FUNCTION_BLOCK Matrix_Inverse (* Template for a simple Basic Function Block Type *)
  (* Standard: 61499-2; Description: Calculates an Inverse of a matrix useing Gauss Jordan Elimination Method. *)
  (* Version 1.0, 2020-08-06, Hafiezd *)
  (* Version 1.1, 2020-08-12, Candra Wardaya *)
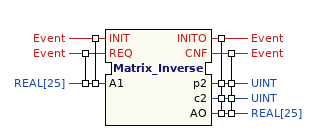
  EVENT_INPUT
    INIT WITH A1; (* Initialization Request *)
    REQ WITH A1; (* Normal Execution Request *)
  END_EVENT
  EVENT_OUTPUT
    INITO WITH AO, p2, c2; (* Initialization Confirm *)
    CNF WITH AO, p2, c2; (* Execution Confirmation *)
  END_EVENT
  VAR_INPUT
    A1 : ARRAY [0..24] OF REAL; (* Matrix Array Input *)
  END_VAR
  VAR_OUTPUT
    p2 : UINT; (* Output Row Size *)
    c2 : UINT; (* Output Column Size *)
    AO : ARRAY [0..24] OF REAL; (* Matrix Inverse Output Array *)
  END_VAR
  VAR
    i : UINT; (* Row Index *)
    j : UINT; (* Column Index *)
    c1 : UINT; (* Augmented Column Size *)
    B : ARRAY [0..99] OF REAL; (* Augmented Matrix of p * c_aug size *)
    ratio : REAL; (* zero-ing factor *)
    k : UINT; (* Augmented Column Index *)
    divisor : REAL; (* Identity factor *)
    p : UINT := 5; (* Internal Variable *)
    c : UINT := 5; (* Internal Variable *)
  END_VAR
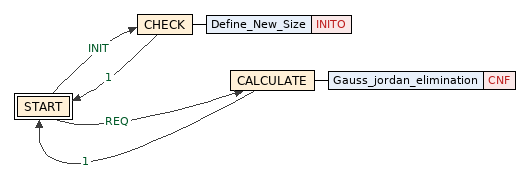
  EC_STATES
    START; (* Initial State *)
    CHECK : Define_New_Size -> INITO;
    CALCULATE : Gauss_jordan_elimination -> CNF;
  END_STATES
  EC_TRANSITIONS
    START TO CHECK := INIT;
    CHECK TO START := 1;
    START TO CALCULATE := REQ;
    CALCULATE TO START := 1;
  END_TRANSITIONS
  ALGORITHM Define_New_Size IN ST: (* new algorithm *)
c2 := c;
p2 := p;
c1 := c*2;
  END_ALGORITHM
  ALGORITHM Gauss_jordan_elimination IN ST: (* new algorithm *)
for i :=1 to c by 1 do  																								/*Start Matrix augmentation */

	for j :=1 to c1 by 1 do

		if i =1 AND j <=c then
			B[c1*i+j-(c1+1)] := A1[c1*i+j-(c1+1)];  //input nilai

		elsif i >1 AND j <=c then
			B[c1*i+j-(c1+1)] := A1[c1*i+j-(c1+1)-(i-1)*(c1-c)];

		else
		// matrix identitas
			if i = j-c then
				B[c1*i+j-(c1+1)] := 1;
			else
				B[c1*i+j-(c1+1)] := 0;
			end_if;

		end_if;

	end_for;

end_for; 																													/*End Matrix augmentation */

for i := 1 to c by 1 do 																								/*Start Gauss Jordan Elimination */
	for j := 1 to c by 1 do
		if i <> j then
			ratio := B[(j-1)*c1+(i-1)] / B[i*c1-c1+i-1];

			for k := 1 to c1 by 1 do
				B[c1*j+k-(c1+1)] := B[c1*j+k-(c1+1)] - ratio * B[c1*i+k-(c1+1)];
			end_for;

		end_if;
	end_for;
end_for; 																													/*End Gauss Jordan Elimination */

for i := 1 to c by 1 do 																								/*Start Row Operation */
	divisor := B[i*c1-c1+(i-1)];

	for j := 1 to c1 by 1 do
		B[c1*i+j-(c1+1)] := B[c1*i+j-(c1+1)] / divisor;
	end_for;

end_for; 																													/*End Row Operation */

for i := 1 to p2 by 1 do 																							/*Output Matrix Inverse Mapping*/

	for j := 1 to c2 by 1 do
		AO[c2*i+j-(c2+1)] := B[c2*i+j-(c2+1)+c2*i];
	end_for;

end_for;
  END_ALGORITHM
END_FUNCTION_BLOCK
